{attribute 'GeneratedUsingTerminal: EL9410-0000-0016'}
{attribute addProperty BoxType "EL9410-0000-0016"}
{attribute addProperty Id "UndervoltageAT %I*BOOL1"}
{attribute addProperty CRC "2984778146"}
{attribute addProperty Size "1"}
TYPE Status_Up_B1E819A2 :
STRUCT
	{attribute addProperty Name "Undervoltage"}
	Undervoltage AT %I* : BOOL;
END_STRUCT
END_TYPE

(* stored: Version 1.2.0.0, ProductVersion 3.1.4024.9
   DUT Status_Up_B1E819A2: Id {d1fa3b8e-fc63-452a-8000-a765f0811772} *)
